{attribute 'qualified_only'}

VAR_GLOBAL CONSTANT
    FILL_TIMEOUT    : TIME := T#15S;  
    FILL_DONE_DELAY : TIME := T#1S;
    RESUME_DELAY    : TIME := T#3S;   
    SETTLE_DELAY    : TIME := T#500MS; 
    BOTTLE_ARRIVE   : TIME := T#3S;    
    SIM_FILL_TIME   : TIME := T#4S;   
    MAX_BOTTLES     : INT  := 9999;
    ALARM_BLINK     : TIME := T#500MS;
END_VAR

(* stored: Version 1.1.0.1, ProductVersion 3.1.4024.16
   GVL GVL_Constants: Id {b8bd0a90-533c-4b12-9ac9-bd41f87a617b} *)
